(* PLC project mdescent, Dassault Systèmes ControlBuild 2024x *)
(* stored: creationDateTime 2023-10-03T11:13:46-01:00 *)

PROGRAM drill.mdescent
  VAR_INPUT
    slowAscent : BOOL := false;
    fastAscent : BOOL := false;
    slowDescent : BOOL := false;
    fastDescent : BOOL := false;
  END_VAR
  VAR_INPUT
    acknowledgePB : BOOL := false;
  END_VAR
  VAR_INPUT
    autoMode : BOOL := false;
    manualMode : BOOL := false;
  END_VAR
  VAR_OUTPUT
    ascentEnd : BOOL := false;
    topDeceleration : BOOL := false;
    downDeceleration : BOOL := false;
    descentEnd : BOOL := false;
    motorFault : DINT := 0;
  END_VAR

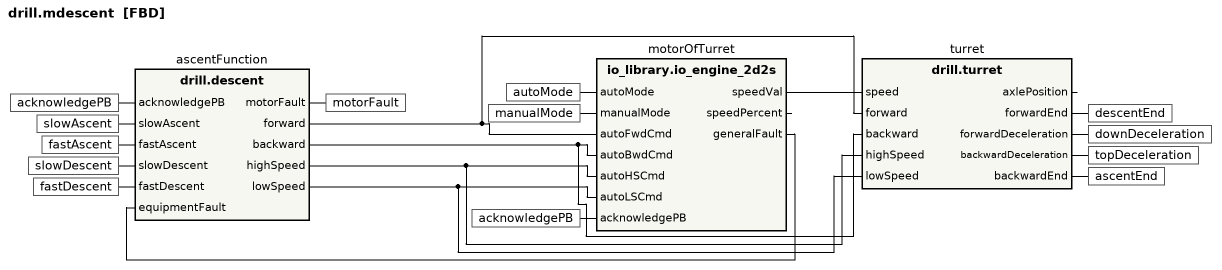
(* FBD diagram, written out as Structured Text *)
motorOfTurret(autoMode := autoMode, manualMode := manualMode, autoFwdCmd := ascentFunction.forward, autoBwdCmd := ascentFunction.backward, autoHSCmd := ascentFunction.highSpeed, autoLSCmd := ascentFunction.lowSpeed, acknowledgePB := acknowledgePB);
ascentFunction(acknowledgePB := acknowledgePB, slowAscent := slowAscent, fastAscent := fastAscent, slowDescent := slowDescent, fastDescent := fastDescent, equipmentFault := motorOfTurret.generalFault);
motorFault := ascentFunction.motorFault;
turret(speed := motorOfTurret.speedVal, forward := ascentFunction.forward, backward := ascentFunction.backward, highSpeed := ascentFunction.highSpeed, lowSpeed := ascentFunction.lowSpeed);
descentEnd := turret.forwardEnd;
downDeceleration := turret.forwardDeceleration;
topDeceleration := turret.backwardDeceleration;
ascentEnd := turret.backwardEnd;
END_PROGRAM
